(* IEC 61131-3 sources: peatyBriquette/Libraries/AsL2DP, 2 files *)

(* ---- AsL2DP.fun ---- *)
(********************************************************************
 * COPYRIGHT (C) BERNECKER + RAINER, AUSTRIA, A-5142 EGGELSBERG
 ********************************************************************
 * Library: AsL2Dp
 * File: AsL2Dp.fun
 * Created: 11.11.2003
 ********************************************************************
 * Functions and function blocks of library AsL2Dp
 ********************************************************************)
FUNCTION_BLOCK L2DPSlave			(*copies output data when received to the output data buffer and sends the input data to the master*)
	VAR_INPUT
		enable	:BOOL;				(*enables execution*)
		device	:UDINT;				(*device name given as a pointer, e.g., ”SLX.SSY”*)
		L2DPid	:UINT;				(*dummy input parameter*)
		outbuf	:UDINT;				(*pointer to the output data area*)
		outlen	:USINT;				(*length of the transferred output data*)
		inbuf	:UDINT;				(*pointer to the input data area*)
		inlen	:USINT;				(*length of the transferred input data*)
		outcopy	:UDINT;				(*pointer to bool, 1/0 = output copying is active/inactive*)
		incopy	:UDINT;				(*pointer to bool, 1/0 = input copying is active/inactive*)
	END_VAR
	VAR_OUTPUT
		status	:UINT;				(*execution status: ERR_OK, ERR_FUB_ENABLE_FALSE, 0xXXXX = see help*)
	END_VAR
	VAR
		init	:USINT;				(*internal variable*)
		byRunState	:USINT;			(*internal variable*)
		baudrate	:USINT;			(*internal variable*)
		diagflag	:USINT;			(*internal variable*)
		pCfgData	:UDINT;			(*internal variable*)
		pInData	:UDINT;				(*internal variable*)
		pDiagData	:UDINT;		    (*internal variable*)
		param0	:UDINT;				(*internal variable*)
		param4	:UDINT;				(*internal variable*)
		param8	:UDINT;				(*internal variable*)
		param12	:UDINT;				(*internal variable*)
		param16	:UDINT;				(*internal variable*)
		param20	:UDINT;				(*internal variable*)
		base0	:UDINT;				(*internal variable*)
		base1	:UDINT;				(*internal variable*)
		base2	:UDINT;				(*internal variable*)
		base3	:UDINT;				(*internal variable*)
		base4	:UDINT;				(*internal variable*)
		base5	:UDINT;				(*internal variable*)
		base6	:UDINT;				(*internal variable*)
		base7	:UDINT;				(*internal variable*)
		base8	:UDINT;				(*internal variable*)
		base9	:UDINT;				(*internal variable*)
		base10	:UDINT;				(*internal variable*)
		base11	:UDINT;				(*internal variable*)
		base12	:UDINT;				(*internal variable*)
		base13	:UDINT;				(*internal variable*)
		base14	:UDINT;				(*internal variable*)
		base15	:UDINT;				(*internal variable*)
		base16	:UDINT;				(*internal variable*)
		base17	:UDINT;				(*internal variable*)
		base18	:UDINT;				(*internal variable*)
		base19	:UDINT;				(*internal variable*)
		base20	:UDINT;				(*internal variable*)
		base21	:UDINT;				(*internal variable*)
		base22	:UDINT;				(*internal variable*)
		base23	:UDINT;				(*internal variable*)
		base24	:UDINT;				(*internal variable*)
		base25	:UDINT;				(*internal variable*)
	END_VAR
END_FUNCTION_BLOCK

(* ---- AsL2DP.var ---- *)
(********************************************************************
 * COPYRIGHT (C) BERNECKER + RAINER, AUSTRIA, A-5142 EGGELSBERG
 ********************************************************************
 * Library: AsL2Dp
 * File: AsL2Dp.var
 * Created: 11.11.2003
 ********************************************************************
 * Constants of library AsL2Dp
 ********************************************************************)
VAR CONSTANT
	ERR_ASL2DP_WAIT_FOR_DATAMODE	: UINT	:= 28826;	(*data transfermode is not jet reached*)
	ERR_ASL2DP_WRONG_OUTDATAPTR	: UINT	:= 28821;		(*0 = output data pointer and 0 != output data length*)
	ERR_ASL2DP_WRONG_DESCRIPTOR	: UINT	:= 28820;		(*string "SLx.SSy" not valid*)
	ERR_ASL2DP_WRONG_SUBSLOTNR	: UINT	:= 28822;		(*determined slot on the module is not supported*)
	ERR_ASL2DP_WRONG_INDATAPTR	: UINT	:= 28823;		(*0 = input data pointer and 0 != input data length*)
	ERR_ASL2DP_WRONG_MODULTYP	: UINT	:= 28825;		(*no L2DP slave module*)
	ERR_ASL2DP_INIT_LESS_MEM	: UINT	:= 28827;		(*L2DP has too less memory*)
	ERR_ASL2DP_WRONG_SLOTNR	: UINT	:= 28824;			(*determined module is not present*)
	ERR_ASL2DP_DP_STATE	: UINT	:= 28828;				(*internal statemaschine error*)
	ERR_ASL2DP_INDATA_TOOLONG	: UINT	:= 28831;		(*maximum input datalength exceeded*)
	ERR_ASL2DP_IO_DATA_TOOLONG	: UINT	:= 28832;		(*maximum output and input datalength exceeded*)
	ERR_ASL2DP_OUTDATA_TOOLONG	: UINT	:= 28830;		(*maximum output datalength exceeded*)
	ERR_ASL2DP_WRONG_NODENR	: UINT	:= 28829;			(*invalid node number*)
	ASL2DP_MAX_INPUTLENGTH	: USINT	:= 240;				(*maximum data length (input direction)*)
	ASL2DP_MAX_IN_OUT_LENGTH	: UINT	:= 368;			(*maximum data length*)
	ASL2DP_MAX_OUTPUTLENGTH	: USINT	:= 240;				(*maximum data length (output direction)*)
	ASL2DP_VPC3_MAX_INPUTLENGTH	: USINT	:= 244;			(*maximum data length (input direction) - VPC3*)
	ASL2DP_VPC3_MAX_IN_OUT_LENGTH	: UINT	:= 488;		(*maximum data length - VPC3*)
	ASL2DP_VPC3_MAX_OUTPUTLENGTH	: USINT	:= 244;		(*maximum data length (output direction) - VPC3*)
END_VAR
